TYPE E_LaudaParameterReadState :
(
	READY,
	ACTUAL_TEMPERATURE_SETPOINT,
	BAH_OUTFLOW_TEMP,
	PUMP_STAGE,
	READ_ENABLE_STATE,
	OIL_LEVEL,
	DONE
);
END_TYPE

(* stored: Version 1.1.0.1, ProductVersion 3.1.4024.12
   DUT E_LaudaParameterReadState: Id {fcbc352a-760d-4356-84af-028413321bce} *)
